FUNCTION TryConvert_SINT_TO_LINT : BOOL
VAR_INPUT
	in : SINT;
	out : REFERENCE TO LINT;
END_VAR

out := SINT_TO_LINT(in);
TryConvert_SINT_TO_LINT := TRUE;

END_FUNCTION

(* stored: Version 1.1.0.1, ProductVersion 3.1.4024.12
   POU TryConvert_SINT_TO_LINT: Id {67387f33-e029-4ea3-9e80-cf0bf989ded5}, SpecialFunc None *)
